{attribute 'qualified_only'}
VAR_GLOBAL
END_VAR

(* stored: Version 1.1.0.1, ProductVersion 3.1.4024.10
   GVL Input: Id {adf02ddf-6e0c-4c19-bbf8-027b47cf2511} *)
